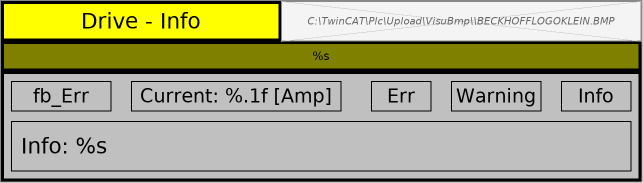
VISUALIZATION Drive_Diag_Info  // 643x183
VAR_IN_OUT
	m_Input_Instance : None;
END_VAR
    Group (1,1 638x178)
        Rectangle (0,70 640x110)
        RoundedRectangle (10,80 100x30), "fb_Err", colour toggle: (Global_Var_AxisInterface.stDrivefunctions[m_Input_Instance].DiagInfobErr) <> 0
        Rectangle (0,0 280x40), "Drive - Info"
        Rectangle (0,40 640x30), "%s", text variable: m_Input_Instance_Str
        Image (280,0 360x40), image: C:\TwinCAT\Plc\Upload\VisuBmp\\BECKHOFFLOGOKLEIN.BMP
        RoundedRectangle (10,120 620x50), "Info: %s", text variable: Global_Var_AxisInterface.stDrivefunctions[m_Input_Instance].stDiagInfo.sMsg
        RoundedRectangle (370,80 60x30), "Err", colour toggle: (Global_Var_AxisInterface.stDrivefunctions[m_Input_Instance].stDiagInfo.bError) <> 0
        RoundedRectangle (450,80 90x30), "Warning", colour toggle: (Global_Var_AxisInterface.stDrivefunctions[m_Input_Instance].stDiagInfo.bWarning) <> 0
        RoundedRectangle (560,80 70x30), "Info", colour toggle: (Global_Var_AxisInterface.stDrivefunctions[m_Input_Instance].stDiagInfo.bInfo) <> 0
        RoundedRectangle (130,80 210x30), "Current: %.1f [Amp]", text variable: Global_Var_AxisInterface.stAxesGlobalVars[m_Input_Instance].fCurrentConsumption
END_VISUALIZATION

(* stored: Version 1.1.0.1, ProductVersion 3.1.4024.11
   Visu Drive_Diag_Info: Id {6bcb564e-c06b-4830-86e3-b2b42e94e332} *)
